% RSLogix 500 project P9_KOBIERSKI_M_v2.RSS, saved by version 8.30.00.16 %
PROJECT "UNTITLED"    % processor: Bul.1763 MicroLogix 1100 Series B %

PROGRAM FILES
  LAD 2 "MAIN"  14 rungs

DATA FILES
  O0 OUTPUT  4 elements
  I1 INPUT  6 elements
  S2 STATUS  66 elements
  B3 BINARY  1 elements
  T4 TIMER  4 elements
  C5 COUNTER  1 elements
  R6 CONTROL  1 elements
  N7 INTEGER  4 elements
  F8 FLOAT  1 elements
  ST9 STRINGS  7 elements

LADDER 2 "MAIN"
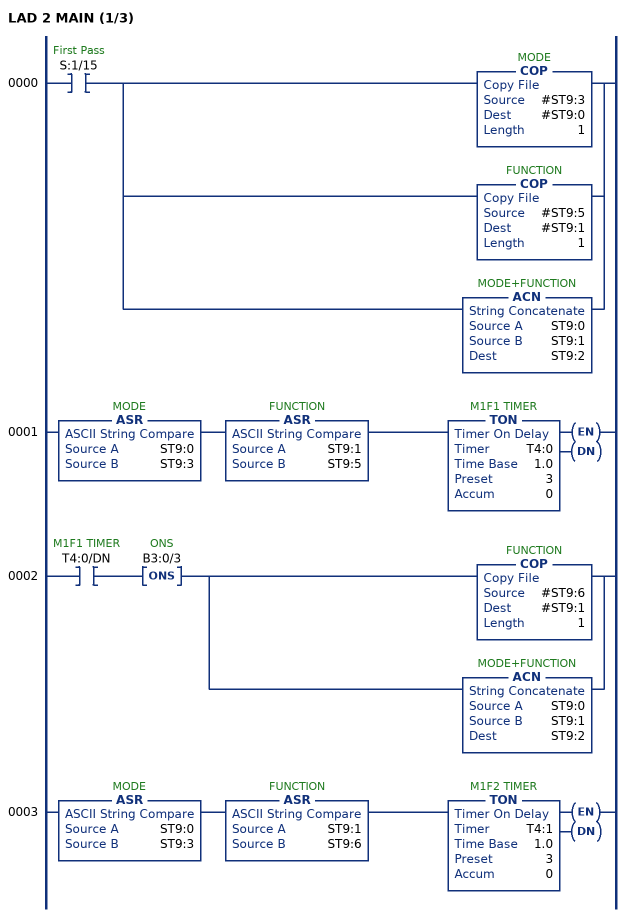
% Rung: 0 %
SOR XIC S:1/15 BST COP #ST9:3 #ST9:0 1 NXB COP #ST9:5 #ST9:1 1 NXB ACN ST9:0 ST9:1 ST9:2 BND EOR
%   S:1/15  "First Pass" %
%   ST9:3  "M1" %
%   ST9:0  "MODE" %
%   ST9:5  "F1" %
%   ST9:1  "FUNCTION" %
%   ST9:2  "MODE+FUNCTION" %
% Rung: 1 %
SOR ASR ST9:0 ST9:3 ASR ST9:1 ST9:5 TON T4:0 1.0 3 0 EOR
%   ST9:0  "MODE" %
%   ST9:3  "M1" %
%   ST9:1  "FUNCTION" %
%   ST9:5  "F1" %
%   T4:0  "M1F1 TIMER" %
% Rung: 2 %
SOR XIC T4:0/DN ONS B3:0/3 BST COP #ST9:6 #ST9:1 1 NXB ACN ST9:0 ST9:1 ST9:2 BND EOR
%   T4:0  "M1F1 TIMER" %
%   B3:0/3  "ONS" %
%   ST9:6  "F2" %
%   ST9:1  "FUNCTION" %
%   ST9:0  "MODE" %
%   ST9:2  "MODE+FUNCTION" %
% Rung: 3 %
SOR ASR ST9:0 ST9:3 ASR ST9:1 ST9:6 TON T4:1 1.0 3 0 EOR
%   ST9:0  "MODE" %
%   ST9:3  "M1" %
%   ST9:1  "FUNCTION" %
%   ST9:6  "F2" %
%   T4:1  "M1F2 TIMER" %

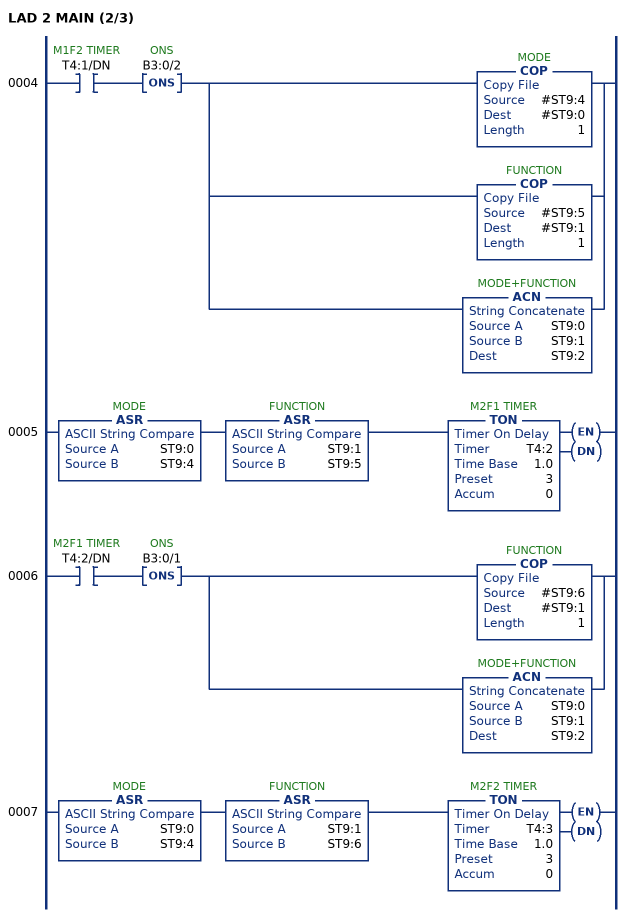
% Rung: 4 %
SOR XIC T4:1/DN ONS B3:0/2 BST COP #ST9:4 #ST9:0 1 NXB COP #ST9:5 #ST9:1 1 NXB ACN ST9:0 ST9:1 ST9:2 BND EOR
%   T4:1  "M1F2 TIMER" %
%   B3:0/2  "ONS" %
%   ST9:4  "M2" %
%   ST9:0  "MODE" %
%   ST9:5  "F1" %
%   ST9:1  "FUNCTION" %
%   ST9:2  "MODE+FUNCTION" %
% Rung: 5 %
SOR ASR ST9:0 ST9:4 ASR ST9:1 ST9:5 TON T4:2 1.0 3 0 EOR
%   ST9:0  "MODE" %
%   ST9:4  "M2" %
%   ST9:1  "FUNCTION" %
%   ST9:5  "F1" %
%   T4:2  "M2F1 TIMER" %
% Rung: 6 %
SOR XIC T4:2/DN ONS B3:0/1 BST COP #ST9:6 #ST9:1 1 NXB ACN ST9:0 ST9:1 ST9:2 BND EOR
%   T4:2  "M2F1 TIMER" %
%   B3:0/1  "ONS" %
%   ST9:6  "F2" %
%   ST9:1  "FUNCTION" %
%   ST9:0  "MODE" %
%   ST9:2  "MODE+FUNCTION" %
% Rung: 7 %
SOR ASR ST9:0 ST9:4 ASR ST9:1 ST9:6 TON T4:3 1.0 3 0 EOR
%   ST9:0  "MODE" %
%   ST9:4  "M2" %
%   ST9:1  "FUNCTION" %
%   ST9:6  "F2" %
%   T4:3  "M2F2 TIMER" %

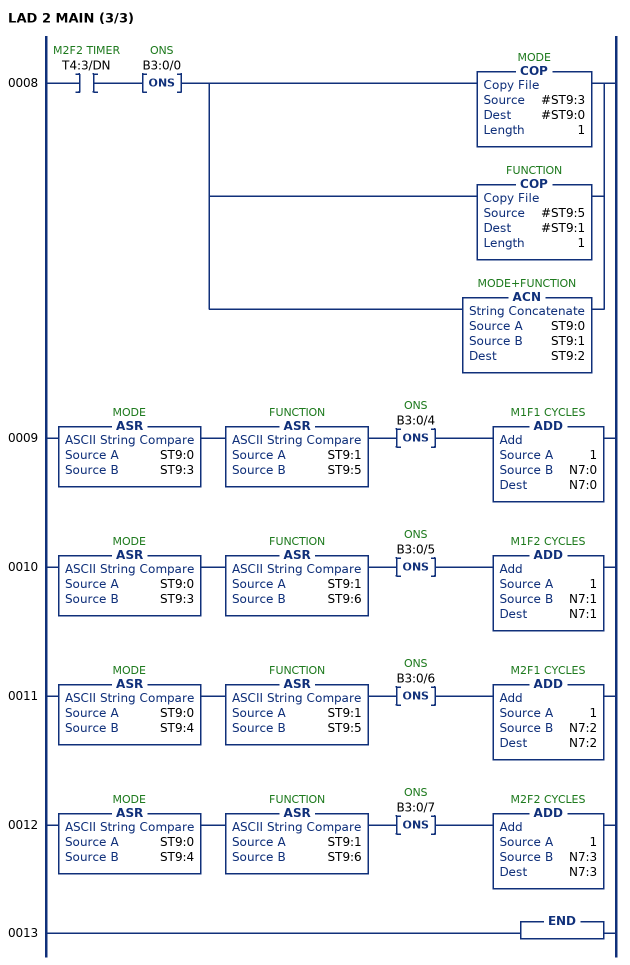
% Rung: 8 %
SOR XIC T4:3/DN ONS B3:0/0 BST COP #ST9:3 #ST9:0 1 NXB COP #ST9:5 #ST9:1 1 NXB ACN ST9:0 ST9:1 ST9:2 BND EOR
%   T4:3  "M2F2 TIMER" %
%   B3:0/0  "ONS" %
%   ST9:3  "M1" %
%   ST9:0  "MODE" %
%   ST9:5  "F1" %
%   ST9:1  "FUNCTION" %
%   ST9:2  "MODE+FUNCTION" %
% Rung: 9 %
SOR ASR ST9:0 ST9:3 ASR ST9:1 ST9:5 ONS B3:0/4 ADD 1 N7:0 N7:0 EOR
%   ST9:0  "MODE" %
%   ST9:3  "M1" %
%   ST9:1  "FUNCTION" %
%   ST9:5  "F1" %
%   B3:0/4  "ONS" %
%   N7:0  "M1F1 CYCLES" %
% Rung: 10 %
SOR ASR ST9:0 ST9:3 ASR ST9:1 ST9:6 ONS B3:0/5 ADD 1 N7:1 N7:1 EOR
%   ST9:0  "MODE" %
%   ST9:3  "M1" %
%   ST9:1  "FUNCTION" %
%   ST9:6  "F2" %
%   B3:0/5  "ONS" %
%   N7:1  "M1F2 CYCLES" %
% Rung: 11 %
SOR ASR ST9:0 ST9:4 ASR ST9:1 ST9:5 ONS B3:0/6 ADD 1 N7:2 N7:2 EOR
%   ST9:0  "MODE" %
%   ST9:4  "M2" %
%   ST9:1  "FUNCTION" %
%   ST9:5  "F1" %
%   B3:0/6  "ONS" %
%   N7:2  "M2F1 CYCLES" %
% Rung: 12 %
SOR ASR ST9:0 ST9:4 ASR ST9:1 ST9:6 ONS B3:0/7 ADD 1 N7:3 N7:3 EOR
%   ST9:0  "MODE" %
%   ST9:4  "M2" %
%   ST9:1  "FUNCTION" %
%   ST9:6  "F2" %
%   B3:0/7  "ONS" %
%   N7:3  "M2F2 CYCLES" %
% Rung: 13 %
SOR END EOR

OTHER DOCUMENTED ADDRESSES
  Q2:0  "JUMP 1"

DATA TABLE (non-zero values as saved)
DATA T4
% .PRE .ACC %
% T4:0 % 3 0
% T4:1 % 3 0
% T4:2 % 3 0
% T4:3 % 3 0
DATA ST9
% ST9:3 % "Mode-1"
% ST9:4 % "Mode-2"
% ST9:5 % "F1"
% ST9:6 % "F2"
